FUNCTION_BLOCK ADD_COLOR (* COLOR Addition *)
  (* Standard: 61131-3 *)
  (* Version 0.0, 2004-12-15, JHC, Rockwell Automation, Converted from SRC format. *)
  (* Compiler header: package fb.rt.plc.math; *)
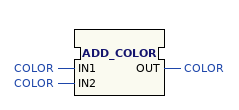
  VAR_INPUT
    IN1 : COLOR; (* Augend *)
    IN2 : COLOR; (* Addend *)
  END_VAR
  VAR_OUTPUT
    OUT : COLOR; (* Sum *)
  END_VAR
END_FUNCTION_BLOCK
